SUBAPPLICATION HebenSenken_QDA_PWM (* Waehlt per 2 AX-Booleans (HEBEN/SENKEN) zwischen 3 ratiometrischen PWM-Stufen (Danfoss PVEA: 25%=Senken, 50%=Neutral, 75%=Heben, Lastteiler-korrigiert) und gibt sie auf einen physischen PWM-Ausgang aus. Reiner Mux+Skalierungs+Ausgabe-Teil von HebenSenken_ILOCK_QDA_PWM_OPC, OHNE Remote-Subscribe/ILOCK/Publish - fuer Aufrufer, die HEBEN/SENKEN bereits anderweitig liefern (z.B. schon gegated/exklusiv, oder wie bei Bunkerboden_PWM nur eine der beiden Richtungen ueberhaupt nutzen, die andere dauerhaft FALSE). Aufrufer muss selbst sicherstellen, dass HEBEN und SENKEN nie gleichzeitig TRUE sind (kein ILOCK hier drin) - sonst liefert AR_AUI_MUX_3 fuer K=3 ein undefiniertes Verhalten. *)
  (* Standard: 61499-2; Description: Copyright (c) 2026 Meisterschulen am Ostbahnhof This program and the accompanying materials are made available under the terms of the Eclipse Public License 2.0 which is available at https://www.eclipse.org/legal/epl-2.0/ SPDX-License-Identifier: EPL-2.0 *)
  (* Version 1.0, 2026-09-27, Franz Höpfinger, Meisterschulen am Ostbahnhof, initial implementation - Mux/Skalierungs/Ausgabe-Teilnetz aus HebenSenken_ILOCK_QDA_PWM_OPC herausgeloest (ASSEMBLE_AB_FROM_AX/AB_TO_AUI/values_50_75_25/AR_AUI_MUX_3/AR_R_MUL_Korrektur/AR_R_MUL_PWM13BIT/AR_TO_AD_NUM/DigitalOutput_PWM), HEBEN/SENKEN jetzt direkte AX-Sockets statt Remote-Subscribe+ILOCK. Erster Aufrufer: Bunkerboden_PWM.SUB (nutzt nur SENKEN=Vollgas, HEBEN dauerhaft FALSE - Konvention 75/Heben ist dort unbenutzt). *)
  PACKAGE MyLib::sys;
  IMPORT logiBUS::io::DQ::logiBUS_DO;
  IMPORT logiBUS::io::DQ::logiBUS_DO_S;
  IMPORT MyLib::sys::const::PWM_Konstanten::PWM_LASTTEILER_KORREKTUR;
  IMPORT MyLib::sys::const::PWM_Konstanten::PWM_13BIT_SKALIERUNG;
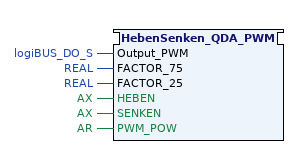
  VAR_INPUT
    Output_PWM : logiBUS::io::DQ::logiBUS_DO_S := logiBUS_DO::Invalid; (* Physischer PWM-Ausgang: 25/50/75% Tastgrad, ratiometrisch *)
    FACTOR_75 : REAL := REAL#1.0; (* Multimeter-kalibrierter Korrekturfaktor auf die nominelle OUT_75-Spanne (25.0), durchgereicht an values_50_75_25.FACTOR_75 - siehe MyLib::sys::const::PWM_Konstanten::VALUES_50_75_25_FACTOR_75 *)
    FACTOR_25 : REAL := REAL#1.0; (* Multimeter-kalibrierter Korrekturfaktor auf die nominelle OUT_25-Spanne (25.0), durchgereicht an values_50_75_25.FACTOR_25 - siehe MyLib::sys::const::PWM_Konstanten::VALUES_50_75_25_FACTOR_25 *)
  END_VAR
  SOCKETS
    HEBEN : adapter::types::unidirectional::AX; (* TRUE waehlt OUT_75 (Heben) - dauerhaft FALSE verdrahten, wenn nicht gebraucht *)
    SENKEN : adapter::types::unidirectional::AX; (* TRUE waehlt OUT_25 (Senken) - dauerhaft FALSE verdrahten, wenn nicht gebraucht *)
    PWM_POW : adapter::types::unidirectional::AR; (* PWM Power 1.0 = Maximale Power, 0.0 = Aus, 0.5 = Halb - durchgereicht an values_50_75_25.PWM_POW *)
  END_SOCKETS
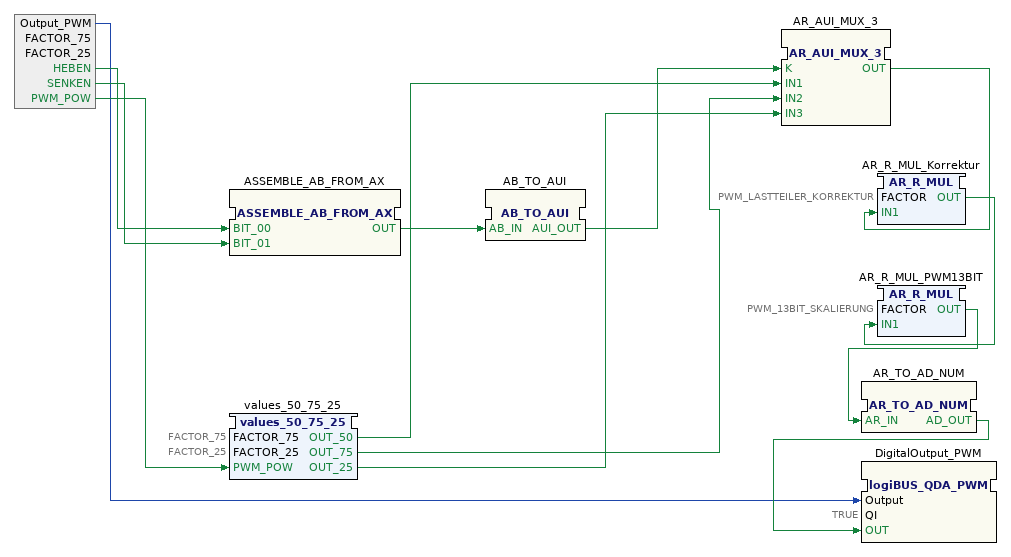
  FBS
    ASSEMBLE_AB_FROM_AX : adapter::assembling::ASSEMBLE_AB_FROM_AX;
    AB_TO_AUI : adapter::conversion::unidirectional::AB_TO_AUI;
    AR_AUI_MUX_3 : adapter::selection::unidirectional::AR_AUI_MUX_3;
    AR_TO_AD_NUM : adapter::conversion::unidirectional::AR_TO_AD_NUM;
    DigitalOutput_PWM : logiBUS::io::DQ::logiBUS_QDA_PWM(QI := TRUE);
  END_FBS
  SUBAPPS
    values_50_75_25 : MyLib::sys::values_50_75_25(FACTOR_75 := FACTOR_75, FACTOR_25 := FACTOR_25);
    AR_R_MUL_Korrektur : MyLib::sys::AR_R_MUL(FACTOR := PWM_LASTTEILER_KORREKTUR);
    AR_R_MUL_PWM13BIT : MyLib::sys::AR_R_MUL(FACTOR := PWM_13BIT_SKALIERUNG);
  END_SUBAPPS
  DATA_CONNECTIONS
    Output_PWM TO DigitalOutput_PWM.Output;
  END_CONNECTIONS
  ADAPTER_CONNECTIONS
    HEBEN TO ASSEMBLE_AB_FROM_AX.BIT_00;
    SENKEN TO ASSEMBLE_AB_FROM_AX.BIT_01;
    ASSEMBLE_AB_FROM_AX.OUT TO AB_TO_AUI.AB_IN;
    AB_TO_AUI.AUI_OUT TO AR_AUI_MUX_3.K;
    PWM_POW TO values_50_75_25.PWM_POW;
    values_50_75_25.OUT_50 TO AR_AUI_MUX_3.IN1;
    values_50_75_25.OUT_75 TO AR_AUI_MUX_3.IN2;
    values_50_75_25.OUT_25 TO AR_AUI_MUX_3.IN3;
    AR_AUI_MUX_3.OUT TO AR_R_MUL_Korrektur.IN1;
    AR_R_MUL_Korrektur.OUT TO AR_R_MUL_PWM13BIT.IN1;
    AR_R_MUL_PWM13BIT.OUT TO AR_TO_AD_NUM.AR_IN;
    AR_TO_AD_NUM.AD_OUT TO DigitalOutput_PWM.OUT;
  END_CONNECTIONS
END_SUBAPPLICATION
